% RSLogix 500 project rev_pulse_code_golf.RSS, saved by version 8.30.00.16 %
PROJECT "UNTITLED"    % processor: Bul.1763 MicroLogix 1100 Series B %

PROGRAM FILES
  LAD 2   2 rungs

DATA FILES
  O0 OUTPUT  4 elements
  I1 INPUT  6 elements
  S2 STATUS  66 elements
  B3 BINARY  24 elements
  T4 TIMER  1 elements
  C5 COUNTER  1 elements
  R6 CONTROL  1 elements
  N7 INTEGER  2 elements
  F8 FLOAT  2 elements

LADDER 2
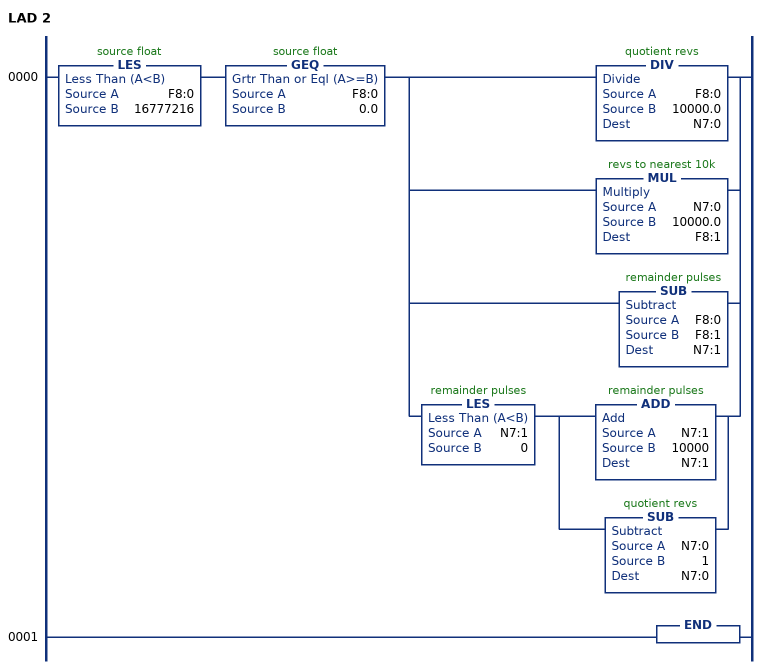
% Rung: 0 %
SOR LES F8:0 16777216 GEQ F8:0 0.0 BST DIV F8:0 10000.0 N7:0 NXB MUL N7:0 10000.0 F8:1 NXB SUB F8:0 F8:1 N7:1 NXB LES N7:1 0 BST ADD N7:1 10000 N7:1 NXB SUB N7:0 1 N7:0 BND BND EOR
%   F8:0  "source float" %
%   N7:0  "quotient revs" %
%   F8:1  "revs to nearest 10k" %
%   N7:1  "remainder pulses" %
% Rung: 1 %
SOR END EOR

OTHER DOCUMENTED ADDRESSES
  B3:0/0  "disable math"
  L9:0  "long pulse count"
  L9:1  "revs"
  L9:2  "remaining pulses"
  L9:3  "working pulse count"
  L9:4  "shifted divisor"
  L9:5  "shifted quotient"
  L9:6  "-1"
  Q2:0  "Monroe ka-chunk"
  S:22  S  "Maximum Observed Scan Time"
